(* CODESYS project SimpleExample

Project tree, tasks and I/O mapping:
  Device : CODESYS Control for Raspberry Pi MC SL, CODESYS GmbH, order no. 2302000009, version 4.9.0.0
  application Application
    libraries: Standard, 3.5.18.0 (System)
    function block Feature [ST]: AlarmRefactor, StartupSequence
    program LocalChange [ST]
    program PLC_PRG [ST]
    program RemotePOU [ST]
    visualisation Visualization
  text list GlobalTextList
  task VISU_TASK (cyclic, interval 100 ms, priority 31) calls VisuElems.Visu_Prg
*)

// Application/Feature
FUNCTION_BLOCK Feature
VAR_INPUT
END_VAR
VAR_OUTPUT
END_VAR
VAR
END_VAR

METHOD AlarmRefactor : BOOL
VAR_INPUT
END_VAR
END_METHOD

METHOD StartupSequence : BOOL
VAR_INPUT
END_VAR
END_METHOD

END_FUNCTION_BLOCK

// Application/LocalChange
PROGRAM LocalChange
VAR
	bTest : BOOL;
	bChange : BOOL;
	bAnotherChange : BOOL;
END_VAR

bTest;

END_PROGRAM

// Application/PLC_PRG
PROGRAM PLC_PRG
VAR
	bTest : REAL;
	bTest2: INT;
	bChange : BOOL;
	bChange2 : BOOL;
	bLocalChange : BOOL;
	bLocalChange2 : BOOL;
	myWorkingBranchChange : BOOL;
	
	VisuText : STRING := 'Hello';
	VisuText1 : STRING := 'Hello1';

END_VAR

myWorkingBranchChange;

END_PROGRAM

// Application/RemotePOU
PROGRAM RemotePOU
VAR
	bTest : bool;
END_VAR

END_PROGRAM

// Application/Visualization
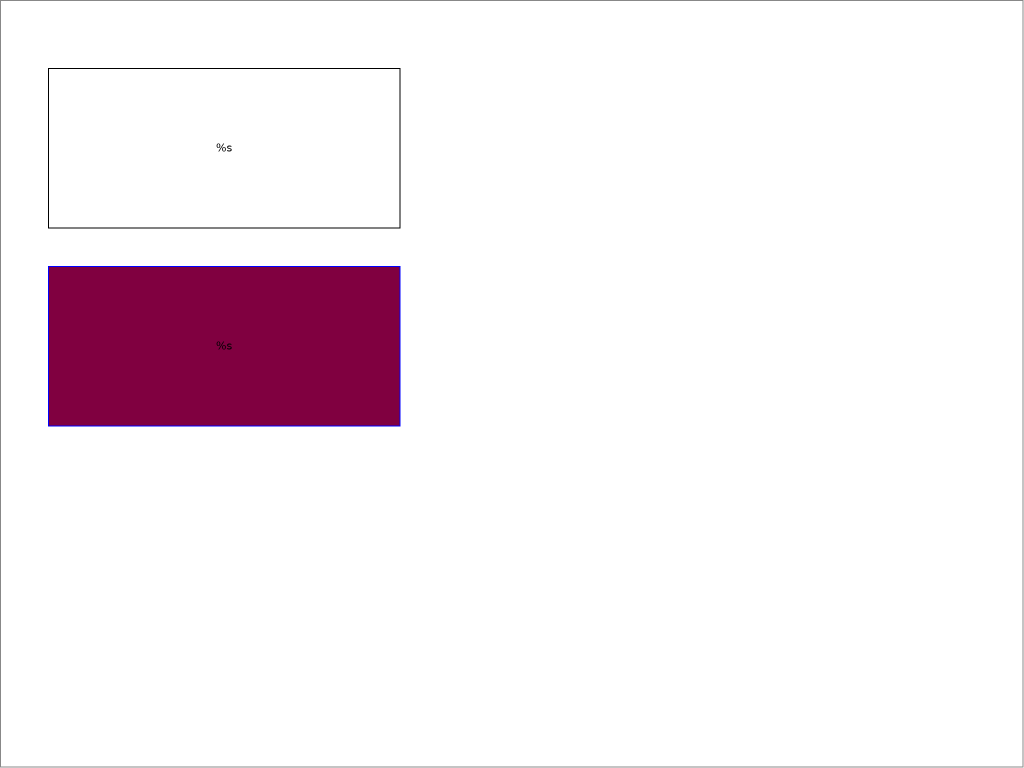
VISUALIZATION Visualization  // 1024x768
    Rectangle (48,68 352x160), "%s", text variable: PLC_PRG.VisuText
    Rectangle (48,266 352x160), "%s", text variable: PLC_PRG.VisuText1
END_VISUALIZATION
